INTERFACE IOutputDevice EXTENDS IDevice

METHOD WriteOutputs
END_METHOD

END_INTERFACE

(* stored: Version 1.1.0.1
   Itf IOutputDevice: Id {bd3d1431-b63c-4fdb-a842-f230bafee062}
   Method WriteOutputs: Id {addcb55a-f6f3-41b2-93ad-709e2fdc7b7d} *)
